{attribute 'linkalways'} 
{attribute 'no_explicit_call' := 'This FB is a CLASS and must be accessed using methods or properties'}
{attribute 'enable_dynamic_creation'}
FUNCTION_BLOCK _ETcVnTemplateMatchMethod EXTENDS EnumDatatypeBase
VAR
	localData : ETcVnTemplateMatchMethod;
	activeData : REFERENCE TO ETcVnTemplateMatchMethod;
	enumBaseDatatype : _DINT(localData);
END_VAR

METHOD PRIVATE AddLocalEnumeration
VAR_INPUT
	Enumeration : T_MAXSTRING;
	Value : ETcVnTemplateMatchMethod;
END_VAR
AddEnumeration(Enumeration, Value);
END_METHOD

PROPERTY PUBLIC Address : PVOID
GET
Address := ADR(activeData);
END_GET
END_PROPERTY

METHOD PUBLIC ClearReference
VAR_INPUT
END_VAR
activeData REF= localData;
SetBaseDatatypeReference();
END_METHOD

METHOD PUBLIC Clone : I_Datatype
VAR
    pClone : POINTER TO _ETcVnTemplateMatchMethod;
END_VAR
pClone := __NEW(_ETcVnTemplateMatchMethod(InitialValue := Value));
Clone := pClone^;
END_METHOD

METHOD FB_init : BOOL
VAR_INPUT
	bInitRetains : BOOL; // if TRUE, the retain variables are initialized (warm start / cold start)
	bInCopyCode : BOOL;  // if TRUE, the instance afterwards gets moved into the copy code (online change)
	InitialValue : ETcVnTemplateMatchMethod;
END_VAR
localData := InitialValue;
AddBaseDatatype(enumBaseDatatype);
ClearReference();

AddLocalEnumeration('TCVN_TMM_SQDIFF', ETcVnTemplateMatchMethod.TCVN_TMM_SQDIFF);
AddLocalEnumeration('TCVN_TMM_SQDIFF_NORMED', ETcVnTemplateMatchMethod.TCVN_TMM_SQDIFF_NORMED);
AddLocalEnumeration('TCVN_TMM_CCORR', ETcVnTemplateMatchMethod.TCVN_TMM_CCORR);
AddLocalEnumeration('TCVN_TMM_CCORR_NORMED', ETcVnTemplateMatchMethod.TCVN_TMM_CCORR_NORMED);
AddLocalEnumeration('TCVN_TMM_CCOEFF', ETcVnTemplateMatchMethod.TCVN_TMM_CCOEFF);
AddLocalEnumeration('TCVN_TMM_CCOEFF_NORMED', ETcVnTemplateMatchMethod.TCVN_TMM_CCOEFF_NORMED);
END_METHOD

PROPERTY PUBLIC Identifier : T_MAXSTRING
GET
Identifier := 'ETcVnTemplateMatchMethod';
END_GET
END_PROPERTY

METHOD IsEnumeratorValueEqual : BOOL
VAR_INPUT
	Enumerator : I_KeyValueForwardEnumerator;
END_VAR
VAR
	storedValue : ETcVnTemplateMatchMethod;
END_VAR
IF NOT Enumerator.TryGet(storedValue) THEN
	RETURN;
END_IF

IsEnumeratorValueEqual := storedValue = activeData;
END_METHOD

METHOD PUBLIC MakeReferenceTo
VAR_INPUT
	ReferenceTarget : REFERENCE TO ETcVnTemplateMatchMethod;
END_VAR
activeData REF= ReferenceTarget;
SetBaseDatatypeReference();
END_METHOD

METHOD PROTECTED SetBaseDatatypeReference
VAR_INPUT
END_VAR
enumBaseDatatype.MakeReferenceTo(activeData);
END_METHOD

PROPERTY PUBLIC Size : UDINT
GET
Size := SIZEOF(activeData);
END_GET
END_PROPERTY

METHOD TryMakeReferenceTo : BOOL
VAR_INPUT
	Target : I_Datatype;
END_VAR
VAR
	targetAsEnum : I_EnumDatatype;
	pTargetData : POINTER TO ETcVnTemplateMatchMethod;
END_VAR
IF NOT Target.TryResolveAsEnumDatatype(targetAsEnum) THEN
	RETURN;
END_IF

IF targetAsEnum.Identifier <> Identifier THEN
	RETURN;
END_IF

pTargetData := Target.Address;
activeData REF= pTargetData^;
SetBaseDatatypeReference();
TryMakeReferenceTo := TRUE;
END_METHOD

PROPERTY PUBLIC Value : ETcVnTemplateMatchMethod
GET
Value := activeData;
END_GET
SET
activeData := Value;
END_SET
END_PROPERTY

END_FUNCTION_BLOCK

(* stored: Version 1.1.0.1
   POU _ETcVnTemplateMatchMethod: Id {fe46ac47-c118-4b81-90f8-e25aa652e7ad}, SpecialFunc None
   Folder Constructor: Id {4b7ba1da-2278-4e8d-9860-a9b6a4ce3d0e}
   Folder Private: Id {08c59cfb-cf51-4819-bb19-bac828f7eee0}
   Folder Protected: Id {450eaa31-89e3-42fb-8662-333f48fa7239}
   Method AddLocalEnumeration: Id {6ab4590f-de3b-4a00-9bee-a06438f36291}
   Property Address: Id {216f1a6f-cd7f-46c5-a2ed-1f41f798d5ec}
   Get Get: Id {c5352690-8f4d-403b-b700-15bd41b0b4b3}
   Method ClearReference: Id {da36dfea-bfdb-426c-8222-00e133fb7bf6}
   Method Clone: Id {fd9f2910-0930-48c8-af44-8a696ec58ade}
   Method FB_init: Id {09df3af6-4605-4a02-9f1e-ef36c6ad8c96}
   Property Identifier: Id {c90cdf67-a014-4712-b9a5-46a52badf8b0}
   Get Get: Id {adf270bd-c71d-4e60-8755-c82dedf4d149}
   Method IsEnumeratorValueEqual: Id {eb53749e-9336-43c8-a120-1d58959efc02}
   Method MakeReferenceTo: Id {9312cf67-5e98-4bb1-8d85-5e726f84d534}
   Method SetBaseDatatypeReference: Id {f70d4726-74af-4a8c-95e1-d2e02374ae78}
   Property Size: Id {2cbd8830-bf12-4c2b-a057-d5a9f13aa2e3}
   Get Get: Id {564919cc-8f3f-4a27-ad6b-66727985f355}
   Method TryMakeReferenceTo: Id {70b55d7e-6e6a-401c-b29b-41a0fb81b1b5}
   Property Value: Id {cedabfc5-4b14-4e51-8028-b23c4f30ef7d}
   Get Get: Id {693cc69f-d815-4549-8a0c-7cbe51093f7c}
   Set Set: Id {0ca00dfa-4546-476e-899c-66da9c827500} *)
